Staubli VAL3: logThrottleMsg.pgx

public program logThrottleMsg(ThrottleLogMsg& x_throttle_msg)
  local num current_time
begin
  // Copyright 2025 ICUBE Laboratory, University of Strasbourg
  //
  // Licensed under the Apache License, Version 2.0 (the "License");
  // you may not use this file except in compliance with the License.
  // You may obtain a copy of the License at
  //
  //     http://www.apache.org/licenses/LICENSE-2.0
  //
  // Unless required by applicable law or agreed to in writing, software
  // distributed under the License is distributed on an "AS IS" BASIS,
  // WITHOUT WARRANTIES OR CONDITIONS OF ANY KIND, either express or implied.
  // See the License for the specific language governing permissions and
  // limitations under the License.

  // Get current time
  current_time = clock()

  // Default severity to INFO
  if (x_throttle_msg.nSeverity == 0)
    x_throttle_msg.nSeverity = 1
  endIf

  // Log the content of a ThrottleMsg
  x_throttle_msg.nMsgCountSinceLastLog = x_throttle_msg.nMsgCountSinceLastLog + 1
  if ((current_time - x_throttle_msg.nLastLogTime) >= x_throttle_msg.nThrottleInterval)
    x_throttle_msg.nLastLogTime = current_time
    logMsg(x_throttle_msg.sMsg + " (msg throttled every " + toString("0.1", x_throttle_msg.nThrottleInterval) + " s, " + toString("0.1", x_throttle_msg.nMsgCountSinceLastLog) + " messages since last log)", x_throttle_msg.nSeverity)
    x_throttle_msg.nMsgCountSinceLastLog = 0
  endIf
end
